// TwinCAT 3 PLC project PLC1
// ProgramVersion: 3.1.4023.0
// libraries:
//   Tc2_Standard, * (Beckhoff Automation GmbH)
//   Tc2_System, * (Beckhoff Automation GmbH)
//   Tc3_Module, * (Beckhoff Automation GmbH)
// project tree:
//   / PlcTask.TcTTO
//   POUs/ MAIN.TcPOU, P_SingleADSRead.TcPOU
// real-time tasks:
//   TASK PlcTask: cycle T#10ms, priority 20, ADS port 350

CONFIGURATION PLC1
    RESOURCE PLC ON TwinCAT3
        TASK PlcTask(INTERVAL := T#10ms, PRIORITY := 20);
        PROGRAM MAIN WITH PlcTask : MAIN;
    END_RESOURCE
END_CONFIGURATION

// ---- POUs/MAIN.TcPOU
PROGRAM MAIN
VAR

END_VAR

P_SingleADSRead();

END_PROGRAM

// ---- POUs/P_SingleADSRead.TcPOU
PROGRAM P_SingleADSRead
VAR
	fbADSRead 		: Tc2_System.ADSREAD;
	sNetId			: Tc2_System.T_AmsNetID := '192.168.10.9.1.1';
	sPort			: Tc2_System.T_AmsPort 	:= 851;
	bRead			: BOOL;
	bReadBool		: BOOL;
	iVarDest		: INT;
	iVarDestBool	: BOOL;
END_VAR

fbADSRead(
	NETID:= sNetId, 
	PORT:= sPort, 
	IDXGRP:= 16#4020, 
	IDXOFFS:= 385000, 
	LEN:= SIZEOF(iVarDest), 	// Tamanho da variável de destino	
	DESTADDR:= ADR(iVarDest), 	// Endereço da variável de destino 
	READ:= bRead, 
	TMOUT:= T#2S, 
	BUSY=> , 
	ERR=> , 
	ERRID=> );
	
fbADSRead(
	NETID:= sNetId, 
	PORT:= sPort, 
	IDXGRP:= 16#4020, 
	IDXOFFS:= 385027, 
	LEN:= SIZEOF(iVarDestBool), 	// Tamanho da variável de destino	
	DESTADDR:= ADR(iVarDestBool), 	// Endereço da variável de destino 
	READ:= bReadBool, 
	TMOUT:= T#2S, 
	BUSY=> , 
	ERR=> , 
	ERRID=> );

END_PROGRAM
